Staubli VAL3: ROBERT_TP6_APPL.dtx

jointRx jStart = {j1=-14.856093, j2=-5.759638, j3=112.561882, j5=73.197755, j6=40.143907}
tool tTool = {fatherId=flange[0], ioLink=valve1}
mdesc mRapide100 = {vel=10}
sio sData = {link=Socket\staubli_server}
bool bAcquisitionOk
pointRx pTarget[3]
  [0] = {x=500, y=-40, z=200, ry=-180, rz=55, fatherId=world[0]}
  [1] = {x=841.429687, y=-222.495582, z=201.936773, rx=-3.5E-05, ry=179.999782, rz=90, fatherId=world[0]}
  [2] = {x=527.606816, y=-37.435701, z=-337.358335, rx=180, rz=-90, fatherId=world[0]}
bool bPinceOpen
pointRx pTemp = {x=527.607274, y=-37.435568, z=403.090503, ry=179.999854, rz=89.999841, fatherId=world[0]}
